TYPE HMIToPLCOperatingMode :
STRUCT
	Manuel	:	HMIActionState;
	Automatic	:	HMIActionState;
	AutomaticStart	:	HMIActionState;
	AutomaticStop	:	HMIActionState;
	Quit	:	HMIActionState;
	Reset	:	HMIActionState;
END_STRUCT
END_TYPE

(* stored: Version 1.1.0.1
   DUT HMIToPLCOperatingMode: Id {2cd37992-3564-4b6e-aab2-dc17be334d75} *)
